% RSLogix 500 project HOURMETER_BAK006.RSS, saved by version 8.30.00.16 %
PROJECT "UNTITLED"    % processor: Bul.1763 MicroLogix 1100 Series B %

PROGRAM FILES
  LAD 2   8 rungs

DATA FILES
  O0 OUTPUT  4 elements
  I1 INPUT  6 elements
  S2 STATUS  66 elements
  B3 BINARY  1 elements
  T4 TIMER  1 elements
  C5 COUNTER  1 elements
  R6 CONTROL  1 elements
  N7 INTEGER  6 elements
  F8 FLOAT  1 elements

LADDER 2
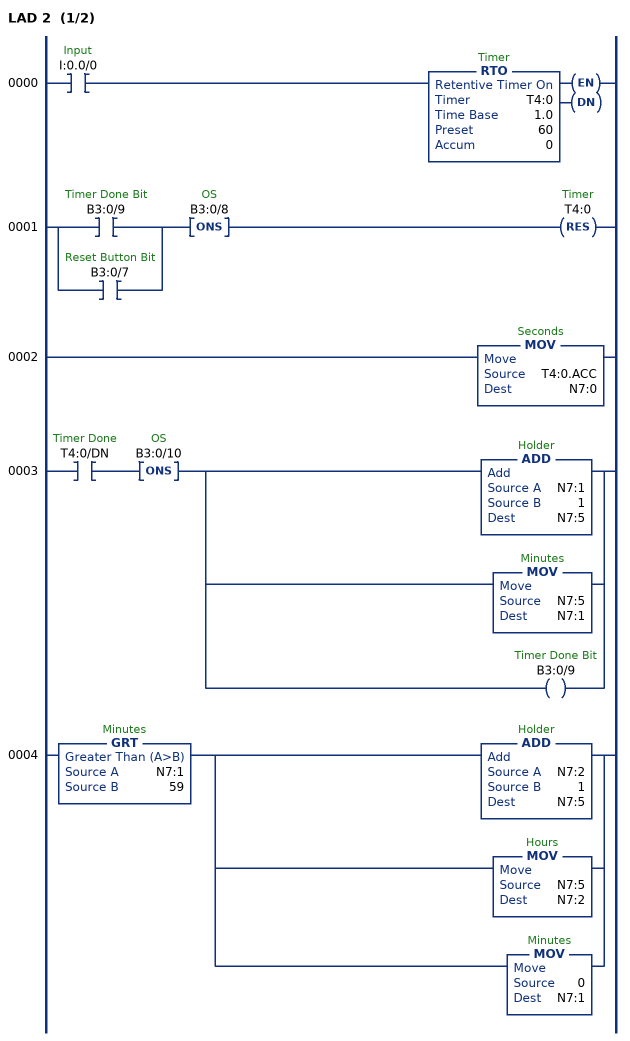
% Rung: 0 %
SOR XIC I:0.0/0 RTO T4:0 1.0 60 0 EOR
%   I:0.0/0  "Input" %
%   T4:0  "Timer" %
% Rung: 1 %
SOR BST XIC B3:0/9 NXB XIC B3:0/7 BND ONS B3:0/8 RES T4:0 EOR
%   B3:0/9  "Timer Done Bit" %
%   B3:0/7  "Reset Button Bit" %
%   B3:0/8  "OS" %
%   T4:0  "Timer" %
% Rung: 2 %
SOR MOV T4:0.ACC N7:0 EOR
%   T4:0.ACC  "Seconds" %
%   N7:0  "Seconds" %
% Rung: 3 %
SOR XIC T4:0/DN ONS B3:0/10 BST BST ADD N7:1 1 N7:5 NXB MOV N7:5 N7:1 BND NXB OTE B3:0/9 BND EOR
%   T4:0/DN  "Timer Done" %
%   B3:0/10  "OS" %
%   N7:1  "Minutes" %
%   N7:5  "Holder" %
%   B3:0/9  "Timer Done Bit" %
% Rung: 4 %
SOR GRT N7:1 59 BST BST ADD N7:2 1 N7:5 NXB MOV N7:5 N7:2 BND NXB MOV 0 N7:1 BND EOR
%   N7:1  "Minutes" %
%   N7:2  "Hours" %
%   N7:5  "Holder" %

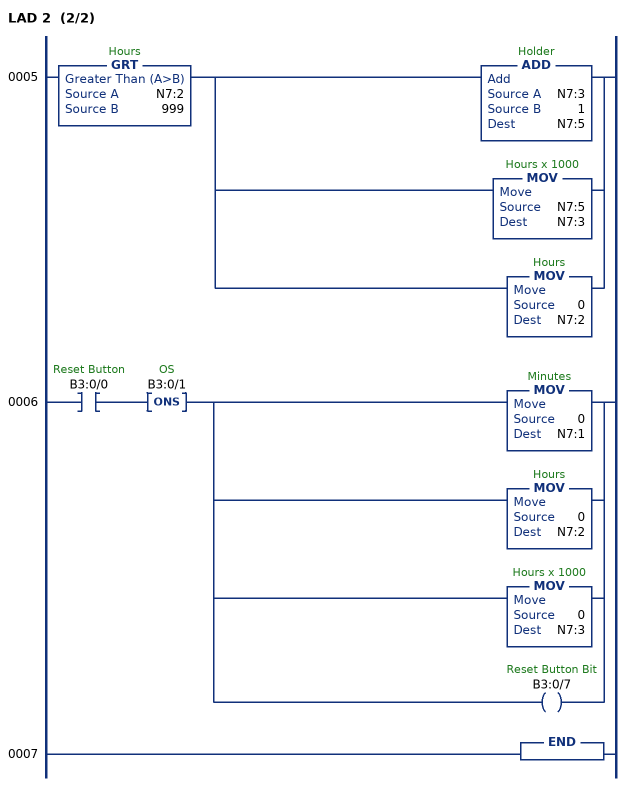
% Rung: 5 %
SOR GRT N7:2 999 BST BST ADD N7:3 1 N7:5 NXB MOV N7:5 N7:3 BND NXB MOV 0 N7:2 BND EOR
%   N7:2  "Hours" %
%   N7:3  "Hours x 1000" %
%   N7:5  "Holder" %
% Rung: 6 %
SOR XIC B3:0/0 ONS B3:0/1 BST MOV 0 N7:1 NXB BST MOV 0 N7:2 NXB BST MOV 0 N7:3 NXB OTE B3:0/7 BND BND BND EOR
%   B3:0/0  "Reset Button" %
%   B3:0/1  "OS" %
%   N7:1  "Minutes" %
%   N7:2  "Hours" %
%   N7:3  "Hours x 1000" %
%   B3:0/7  "Reset Button Bit" %
% Rung: 7 %
SOR END EOR

OTHER DOCUMENTED ADDRESSES
  B3:0/2  "Timer Reset"
  B3:0/3  "OS"
  B3:0/4  "Trigger"
  B3:0/5  "Process Run"
  B3:0/6  "Process Reset"

DATA TABLE (non-zero values as saved)
DATA T4
% .PRE .ACC %
% T4:0 % 60 0
